{attribute 'qualified_only'}
VAR_GLOBAL
END_VAR

(* stored: Version 1.1.0.1, ProductVersion 3.1.4024.16
   GVL Global: Id {5aecde8c-e2e9-44d1-b781-b336d476c435} *)
